FUNCTION_BLOCK FB_MasterFriciton
VAR_INPUT
END_VAR
VAR_OUTPUT
END_VAR
VAR
	// joint friction compensation scale
	m_frictionCompScale :Vec7d :=[0.7, 0.5, 0.5, 0.0, 0.7, 0.7, 0.7];
	
	// joint velocity threshold for coulomb friction transition
	m_cFrictionVelThres : LREAL := 5.0 * g_deg2Rad;
	
	// arm index
	m_armIdx: INT ;
	
	// joint coulomb friction parameters: friction = a * gravityTrq + b;
	m_frictionParamA : Vec7d := g_zeroVec7d;
	m_frictionParamB : Vec7d := g_zeroVec7d;
	
	// joint damping
	m_jntDamp :Vec7d := g_zeroVec7d;
	
	// max joint friciton 
	m_maxFriction :Vec7d;
	

END_VAR

METHOD init : BOOL
VAR_INPUT
	i_armIdx :INT;
END_VAR

VAR
	i:int;
END_VAR
m_armIdx := i_armIdx;

m_frictionParamA := g_zeroVec7d;
m_frictionParamB := g_zeroVec7d;
m_jntDamp := g_zeroVec7d;
m_maxFriction := GVL_ArmDynamics.g_maxJntFriction;

FOR i:=1 TO 7 DO
	m_frictionParamA[i] := GVL_ArmDynamics.g_jntFrictionParam[m_armIdx, 2*i-1];
	m_frictionParamB[i] := GVL_ArmDynamics.g_jntFrictionParam[m_armIdx, 2*i];
END_FOR
END_METHOD

METHOD run : vec7d
VAR_IN_OUT CONSTANT
	// joint gravity torque
	i_jntGravity :Vec7d;
	
	// joint velocity
	i_jntVel :Vec7d;
END_VAR

VAR
	i:INT;
	transitScale:LREAL;
	cFriction, dFriction :LREAL;
END_VAR
FOR i:=1 TO g_mJntNum DO
	transitScale := LIMIT(0, ABS(i_jntVel[i]/m_cFrictionVelThres),1);
	cFriction:=m_frictionParamA[i]*ABS(i_jntGravity[i])+m_frictionParamB[i];
	cFriction:= transitScale * sign(i_jntVel[i]) * cFriction;
	
	dFriction:= i_jntVel[i] * m_jntDamp[i];
	
	run[i] := LIMIT(-m_maxFriction[i], m_frictionCompScale[i] * (cFriction+dFriction) ,m_maxFriction[i]);
END_FOR
END_METHOD

END_FUNCTION_BLOCK

(* stored: Version 1.1.0.1, ProductVersion 3.1.4024.12
   POU FB_MasterFriciton: Id {e1c0a847-1949-4788-8871-72ab788e2df1}, SpecialFunc None
   Method init: Id {6c66ea74-5b37-4c40-853c-a414ffc369f7}
   Method run: Id {0e064868-95f9-4591-a903-e34a876d9e26} *)
